// TIA Portal V19 export
TYPE "HU_Tank_Par"
// stored: Access Published
   STRUCT
      DelayCheckFilterClogged { S7_SetPoint := 'True'} : Time;
      DelayRecirculationPumpOff { S7_SetPoint := 'True'} : Time;
      HeatingEnable { S7_SetPoint := 'True'} : Bool;
      HeatingTempRunPermit { S7_SetPoint := 'True'} : Real;
      HeatingSetpoint { S7_SetPoint := 'True'} : Real;
      HeatingUnit2Delta { S7_SetPoint := 'True'} : Real;
      CoolingEnable { S7_SetPoint := 'True'} : Bool;
      CoolingSetpoint { S7_SetPoint := 'True'} : Real;
      WeeklyClockEnable { S7_SetPoint := 'True'} : Bool;
      WeeklyClockSetup { S7_SetPoint := 'True'} : Array[1..7] of "WkClockSet";
   END_STRUCT;
END_TYPE
